TYPE ST_CyStatus ://
STRUCT
	ONState:	        BOOL;//开状态
	OFFState:	        BOOL;//关状态
	Error1:	            BOOL;//气缸ON报警
	Error2:	            BOOL;//气缸OFF报警
    Errorcomp                   :BOOL; //手自动对 比报警
END_STRUCT
END_TYPE

(* stored: Version 1.1.0.1, ProductVersion 3.1.4024.12
   DUT ST_CyStatus: Id {740c4c8e-fa67-4e17-b84f-758471c1c530} *)
